// Minimal Unit for §7.6.1 tests: owns one basic cylinder, routes manual commands.
FUNCTION_BLOCK FB_ProbeUnitManual EXTENDS FB_UnitBase
VAR_OUTPUT
    Cyl : FB_ConfigurableCylinderCM;
    Hal : ST_ConfigurableCylinderHal;
    Intlk : FB_PermIntlk;
END_VAR

Cyclic();

METHOD Setup : BOOL
VAR_INPUT
    Name : STRING(80);
END_VAR
_M_SetName(Name);
Cyl.Setup(Name := CONCAT(Name, '.Cyl'), HalRef := Hal, Recipe := 0);
Intlk.Define(Index := 1, Description := 'project.interlock.airPressureOk', Reason := E_Reason.PERMISSIVE_NOT_MET, Bypassable := FALSE);
Setup := TRUE;
END_METHOD

METHOD PROTECTED _M_Dispatch
_M_Complete();  // trivial sequence
END_METHOD

METHOD PROTECTED _M_RouteManual : BOOL
VAR_INPUT
    TargetPath : STRING(255);
    Value : DINT;
END_VAR
IF TargetPath = CONCAT(_name, '.Cyl') THEN
    _M_RouteManual := Cyl.ManualCommand(Value := Value);
ELSE
    _M_RouteManual := FALSE;
END_IF
END_METHOD

METHOD PROTECTED OnCyclic : DINT
OnCyclic := SUPER^.OnCyclic();
Intlk();
Cyl();
END_METHOD

METHOD PROTECTED _M_AppendInterlocks
VAR_IN_OUT
    Report : ST_ReleaseReport;
END_VAR
Intlk.AppendFailed(SourcePath := _name, Report := Report);
END_METHOD

METHOD SetAir : BOOL
VAR_INPUT
    Ok : BOOL;
END_VAR
Intlk.Cond[1] := Ok;
SetAir := TRUE;
END_METHOD

// Test injection stays inside the owner; callers cannot write through Cyl VAR_OUTPUT.
METHOD TestSetCylinderAbort : BOOL
VAR_INPUT
    Value : BOOL;
END_VAR
Cyl.Abort := Value;
TestSetCylinderAbort := TRUE;
END_METHOD

// test driver: recompute OEE from externally-set accumulators (§8.5.1 pure compute)
METHOD TestOeeCompute : BOOL
_M_OeeCompute();
TestOeeCompute := TRUE;
END_METHOD

METHOD TestSeedOee
VAR_INPUT
    Good : UDINT;
    Nok : UDINT;
    RunMs : UDINT;
    DownMs : UDINT;
    IdleMs : UDINT;
    IdealCycleMs : UDINT;
END_VAR
GoodCount := Good;
NokCount := Nok;
Oee.RunMs := RunMs;
Oee.DownMs := DownMs;
Oee.IdleMs := IdleMs;
Oee.IdealCycleMs := IdealCycleMs;
END_METHOD

END_FUNCTION_BLOCK

(* stored: Version 1.1.0.1, ProductVersion 3.1.4024.12
   POU FB_ProbeUnitManual: Id {b70d8e32-bdb5-4442-86f6-dfc08ed3da9a}, SpecialFunc None
   Method Setup: Id {a0d6323a-1318-45da-a667-a4eabb1308ff}
   Method _M_Dispatch: Id {65b784f2-3cb8-45c4-9d2f-0967fa381126}
   Method _M_RouteManual: Id {fd9bd26d-5208-41b0-a717-76ac266aa5f1}
   Method OnCyclic: Id {43b1f141-bf55-4e98-99fe-e8371696ffd2}
   Method _M_AppendInterlocks: Id {8160ac86-aa62-483d-99e3-c7c748806f90}
   Method SetAir: Id {7d8f8b1e-d9e0-4b80-92d7-94e8d84b3c69}
   Method TestSetCylinderAbort: Id {0344aab3-3364-4374-b543-2968d6e6ae8b}
   Method TestOeeCompute: Id {877a9d73-6071-4e97-991b-805ab45ff83a}
   Method TestSeedOee: Id {fcd405e2-4b0f-47b5-9c5e-1f24daf9a696} *)
